{attribute 'OPC.UA.DA.JobMethod' := 'JobMethode_VerticalMove'}
FUNCTION_BLOCK HRL_RGB_AS_VerticalMoveEncoder
VAR
	AlwaysTrue : BOOL := TRUE;
	// Used for debugging purposes to display InputArguments of method call
	MethodCall_VerticalMove : BOOL := FALSE; // used to store InputArg "MethodCall" from Start() method
	ResetMethodCall	: BOOL := FALSE;
	Direction : BOOL := FALSE;
	EncoderTargetPosition_01 : UDINT;
	EncoderTargetPosition_02 : UDINT;
	TSR : BOOL;
	callCounterStart : ULINT; // counts how many times the Start() method has been called
	callCounterCheckState : ULINT; // counts how many times the CheckState() method has been called
	callCounterAbort : ULINT; // counts how many times the Abort() method has been called
	
	// Variables to determine if a job has been started (Start() method has been called) or finished
	jobRunning : BOOL;
	jobFinished : BOOL;

	// State machine variable
	state : UDINT;
	
	// FB Intatziation Variable
	HRL_RGB_VerticalMoveWithEncoder : AxisControl_Encoder;
END_VAR
	
VAR_INPUT
	ESS: BOOL;
	EncoderStartPosition_01 : UDINT;
	EncoderStartPosition_02 : UDINT;
	TS01 : BOOL;
	TOF_TSR_TIME : TIME;
	AutomaticMode: BOOL;
END_VAR

VAR_OUTPUT
	Motor_Control_01 : BOOL;
	Motor_Control_02 : BOOL;
END_VAR

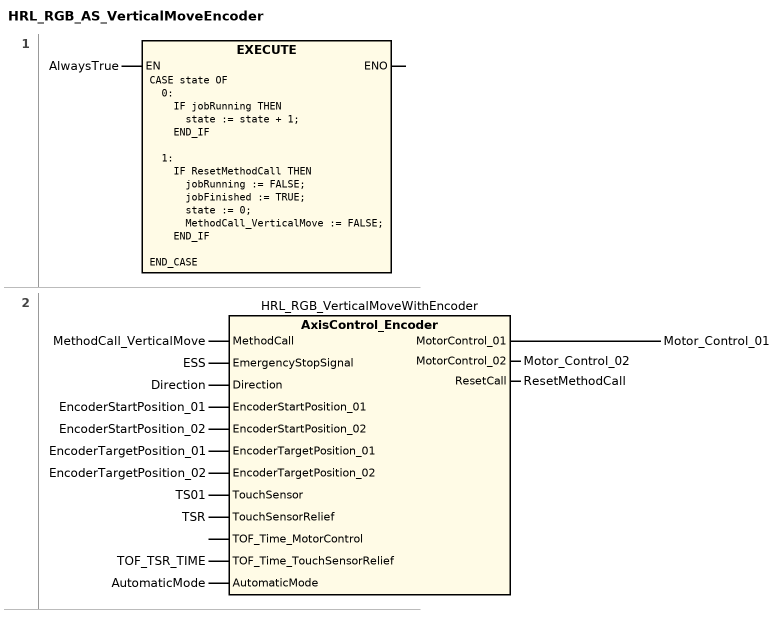
// NETWORK 1
IF AlwaysTrue THEN
    CASE state OF
    	0:
    		IF jobRunning THEN
    			state := state + 1;
    		END_IF
    		
    	1:
    		IF ResetMethodCall THEN
    			jobRunning := FALSE;
    			jobFinished := TRUE;
    			state := 0;
    			MethodCall_VerticalMove := FALSE;
    		END_IF
    		
    END_CASE
END_IF

// NETWORK 2
HRL_RGB_VerticalMoveWithEncoder(
    MethodCall := MethodCall_VerticalMove,
    EmergencyStopSignal := ESS,
    Direction := Direction,
    EncoderStartPosition_01 := EncoderStartPosition_01,
    EncoderStartPosition_02 := EncoderStartPosition_02,
    EncoderTargetPosition_01 := EncoderTargetPosition_01,
    EncoderTargetPosition_02 := EncoderTargetPosition_02,
    TouchSensor := TS01,
    TouchSensorRelief := TSR,
    TOF_Time_TouchSensorRelief := TOF_TSR_TIME,
    AutomaticMode := AutomaticMode,
    MotorControl_02 => Motor_Control_02,
    ResetCall => ResetMethodCall); // AxisControl_Encoder
Motor_Control_01 := HRL_RGB_VerticalMoveWithEncoder.MotorControl_01;

{attribute 'TcRpcEnable' := '1'}
METHOD Abort : HRESULT
VAR_INPUT
	hdl : UDINT; // Do not change, used by server.
END_VAR
callCounterAbort := callCounterAbort + 1;
END_METHOD

{attribute 'TcRpcEnable' := '1'}
METHOD CheckState : HRESULT
VAR_INPUT
	hdl : UDINT; // Do not change, used by server.
END_VAR
VAR_OUTPUT
	bBusy : BOOL; // Do not change. Used by server to find out if the job is finished
	
	// List of OutputArguments for OPC UA method, may be customized
	State : BOOL; // Abgeschlossener MethodCall
	MethodCall: BOOL; //Input Recall
END_VAR
callCounterCheckState := callCounterCheckState + 1;
IF NOT jobFinished THEN
	bBusy := TRUE; // job is not finished yet
	CheckState := 0; // no error
ELSE
	bBusy := FALSE; // job is finished
	CheckState := 0; // done, no error occured during execution (OPC UA StatusCode "GOOD")
	jobFinished := FALSE;
	State := ResetMethodCall;
	MethodCall := MethodCall_VerticalMove;
END_IF
END_METHOD

{attribute 'TcRpcEnable' := '1'}
METHOD Start : HRESULT
VAR_INPUT
	// List of InputArguments for OPC UA method, may be customized
	MethodCall : BOOL; // some description
	MovementDirection : BOOL;
	EncoderPositionVertical_01 : UDINT;
	EncoderPositionVertical_02 : UDINT;
	TouchSensorRelief : BOOL;
END_VAR
VAR_OUTPUT
	hdl : UDINT; // Do not change, used by server.
END_VAR
callCounterStart := callCounterStart + 1;

MethodCall_VerticalMove := MethodCall;
MovementDirection := Direction;
EncoderTargetPosition_01 := EncoderPositionVertical_01;
EncoderTargetPosition_02 := EncoderPositionVertical_02;
TouchSensorRelief := TSR;

jobRunning := TRUE;
Start := 0; // no error occured, e.g. while parsing the input arguments (0 = OPC UA StatusCode "GOOD")
END_METHOD

END_FUNCTION_BLOCK

(* stored: Version 1.1.0.1, ProductVersion 3.1.4024.15
   POU HRL_RGB_AS_VerticalMoveEncoder: Id {fdfb0dc9-c9c2-4773-a117-03f094c5a535}, SpecialFunc None
   Method Abort: Id {b53712c3-6f71-488d-8c27-fc1174a866ca}
   Method CheckState: Id {51b7ed45-46f9-43c0-8594-67bc3ad198d6}
   Method Start: Id {212ae213-5e4c-4cc8-9029-64337fe229be} *)
